DATA_BLOCK "V90Servo_DB"
{ S7_Optimized_Access := 'TRUE' }
VERSION : 0.1
NON_RETAIN
"V90_Servo"

BEGIN

END_DATA_BLOCK

